FUNCTION_BLOCK PreExecutionChecks IMPLEMENTS I_PreExecutionChecks
VAR
	hasFailed : BOOL;
	hasFailedReason : T_MAXSTRING;
END_VAR;

METHOD PUBLIC Fail
VAR_INPUT
	Message : T_MAXSTRING;
END_VAR
IF hasFailed THEN
	RETURN;
END_IF

hasFailed := TRUE;
hasFailedReason := Message;
END_METHOD

PROPERTY PUBLIC Failed : BOOL
GET
Failed := hasFailed;
END_GET
END_PROPERTY

METHOD PUBLIC IsFalse
VAR_INPUT
	Actual : BOOL;
	Message : T_MAXSTRING;
END_VAR
IF hasFailed THEN
	RETURN;
END_IF

IF NOT Actual THEN
	RETURN;
END_IF

hasFailed := TRUE;
hasFailedReason := Message;
END_METHOD

METHOD PUBLIC IsTrue
VAR_INPUT
	Actual : BOOL;
	Message : T_MAXSTRING;
END_VAR
IF hasFailed THEN
	RETURN;
END_IF

IF Actual THEN
	RETURN;
END_IF

hasFailed := TRUE;
hasFailedReason := Message;
END_METHOD

PROPERTY PUBLIC Passed : BOOL
GET
Passed := not hasFailed;
END_GET
END_PROPERTY

PROPERTY PUBLIC Reason : T_MAXSTRING
GET
Reason := hasFailedReason;
END_GET
END_PROPERTY

METHOD PUBLIC Reset
VAR_INPUT
END_VAR
hasFailed := FALSE;
hasFailedReason := '';
END_METHOD

END_FUNCTION_BLOCK

(* stored: Version 1.1.0.1, ProductVersion 3.1.4024.13
   POU PreExecutionChecks: Id {4f154e26-796d-080d-24a3-a63a8f61ff8a}, SpecialFunc None
   Method Fail: Id {0bd7c90c-6f50-0f13-001d-8a21681125d1}
   Property Failed: Id {e294c8a8-8b74-08ab-1d00-60c5721ae57d}
   Get Get: Id {58aceef9-6f7e-02f2-119b-60cda279c115}
   Method IsFalse: Id {c9a51ccb-e070-0fe4-0935-bebcecc81d65}
   Method IsTrue: Id {8f0afc7a-f89f-0972-35c1-5a79962a141d}
   Property Passed: Id {080476fa-4916-0720-298d-b8d0d34d0113}
   Get Get: Id {0f981c83-8beb-0453-070f-53df2356258d}
   Property Reason: Id {bd1454b5-8342-07df-1a61-a42e487082ca}
   Get Get: Id {48fadb59-c617-0c53-3221-f148c2615e9c}
   Method Reset: Id {f111bc43-d56c-0934-0426-37024ae13b4d} *)
